TYPE E_ValueDeviationStatus :
(
	OK,
	NOK
);
END_TYPE

(* stored: Version 1.1.0.1, ProductVersion 3.1.4024.13
   DUT E_ValueDeviationStatus: Id {1c28bd1c-c878-0369-1408-23304e32d7eb} *)
